// TIA Portal V20 export
DATA_BLOCK "ControlNodes"   // DB154
// stored: MemoryReserve 100, Namespace Unit1.Em0
   VAR
      em { ExternalWritable := 'False'} : "LAF_typeEmControlNode";
      cm { ExternalWritable := 'False'} : "Unit1.Em0.typeCmControlNode";
      citiMap : "LER_OEM_Data";
      unWinder { ExternalWritable := 'False'} : "Unit1.Em0.typeSequenceControlNode";
   END_VAR
   VAR RETAIN
      cmUnWinderAxisB { ExternalWritable := 'False'} : "LBC_typeAxisControlNode";
      cmAirShaftOnOff { ExternalWritable := 'False'} : "LBC_typeTwoWayActuatorControlNode";
      cmExpelFwdBwd { ExternalWritable := 'False'} : "LBC_typeTwoWayActuatorControlNode";
      cmTensionCheckSensor { ExternalWritable := 'False'} : "LBC_typeDigitalSignalControlNode";
      cmRadiusMeasureAnalogInput { ExternalWritable := 'False'} : "LBC_typeAnalogInputControlNode";
      cmEpc { ExternalWritable := 'False'} : "LER_typeCON600ControlNode";
      cmRadiusMeasure { ExternalWritable := 'False'} : "LER_typeRadiusMeasureControlNode";
      cmUnWinderAxisB_TorqueCal { ExternalWritable := 'False'} : "LER_typeServoTorqueCalControlNode";
   END_VAR
BEGIN
   // cm.brakeTest.unwinder.monitoring.error : Unwinder Left Axis Brake Test Error
   // cm.brakeTest.unwinder.monitoring.busy : Unwinder Left Axis Brake Test In progress
END_DATA_BLOCK
